INTERFACE I_ProcessController

METHOD HandleIoSignals : BOOL
END_METHOD

END_INTERFACE

(* stored: Version 1.1.0.1, ProductVersion 3.1.4024.9
   Itf I_ProcessController: Id {1cfb29d1-397f-4ea9-bea6-6d38846bc098}
   Method HandleIoSignals: Id {66d611f0-34c7-430b-83e3-199474d0b6be} *)
